TEXTLIST tlNames
  0 = 'Bottle Sensor' | EN: 'Bottle Sensor' | PL: 'Sensor Butelki'
  1 = 'Bottle Eject Sensor' | EN: 'Bottle Eject Sensor' | PL: 'Sensor Wyjazdu Butelki'
  2 = 'Drawer Bottle Sensor' | EN: 'Drawer Bottle Sensor' | PL: 'Sensor Butelki na Szufladzie'
  3 = 'Drawer Lock' | EN: 'Drawer Lock' | PL: 'Zamek Szuflady'
  4 = 'Weight' | EN: 'Weight' | PL: 'Waga'
  5 = 'Out Conveyor' | EN: 'Out Conveyor' | PL: 'Przenosnik Wyjazdowy'
  6 = 'Weighing Actuator' | EN: 'Weighing Actuator' | PL: 'Silownik Wazacy'
  7 = 'Unloading Actuator' | EN: 'Unloading Actuator' | PL: 'Silownik Rozladowujacy'
  8 = 'Pusher Actuator' | EN: 'Pusher Actuator' | PL: 'Silownik Spychajacy'
  9 = 'Separator 1' | EN: 'Separator 1' | PL: 'Separator 1'
  10 = 'Separator 2' | EN: 'Separator 2' | PL: 'Separator 2'
  11 = 'Separator 1 Sensor' | EN: 'Separator 1 Sensor' | PL: 'Separator 1 Czujnik'
  12 = 'Separator 2 Sensor' | EN: 'Separator 2 Sensor' | PL: 'Separator 2 Czujnik'
  13 = 'Table Servo' | EN: 'Table Servo' | PL: 'Table Servo'
   = ''
END_TEXTLIST

(* stored: Version 1.1.0.1, ProductVersion 3.1.4024.16
   TextList tlNames: Id {09652da2-fae6-49b9-9b2a-10e94f8e2354} *)
